PROGRAM MAIN
VAR
	udp1 : UDPConnect;
END_VAR

udp1();

END_PROGRAM

(* stored: Version 1.1.0.1, ProductVersion 3.1.4022.3
   POU MAIN: Id {83da6505-1eb3-48a2-b593-db0aa655616f}, SpecialFunc None *)
